FUNCTION mat3Mat3 : Mat3d
VAR_IN_OUT CONSTANT
	i_mat3a :Mat3d;
	i_mat3b :Mat3d;
END_VAR
VAR
	i,j,k : INT ;
END_VAR

FOR i:=1 TO 3 DO
	FOR j:=1 TO 3 DO
		mat3Mat3[i,j]:=0.0;
		FOR k:=1 TO 3 DO 
		mat3Mat3[i,j]:=mat3Mat3[i,j]+i_mat3a[i,k]*i_mat3b[k,j];
		END_FOR
	END_FOR
END_FOR

END_FUNCTION

(* stored: Version 1.1.0.1, ProductVersion 3.1.4024.12
   POU mat3Mat3: Id {1c07a4d8-5929-4d42-a6ca-15eca4783276}, SpecialFunc None *)
